(* CODESYS project ccssim.library
   Company: ccsim
   Description: CCS simulator library to support testing tracking devices.
   Version: 0.0.2.0
   Placeholder: ESO CCS PLC Simulator Library
   Author: Mario Kiekebusch
   Title: ESO CCS PLC Simulator Library

Project tree, tasks and I/O mapping:
  libraries: ESO LDC Common Library, * (ESO); ESO LDC Timer Library, * (ESO); Tc2_EtherCAT, * (Beckhoff Automation GmbH); Tc2_IoFunctions, * (Beckhoff Automation GmbH); Tc2_Standard, * (Beckhoff Automation GmbH); Tc2_System, * (Beckhoff Automation GmbH); Tc2_Utilities, * (Beckhoff Automation GmbH); Tc3_Module, * (Beckhoff Automation GmbH); VisuDialogs, * (System); ESO ELT Utility Library, * (ESO)
  DUTs/
    Structures/
      data type T_CCS_CFG
      data type T_CCS_CTRL
      data type T_CCS_GUI
      data type T_CCS_STAT
      data type T_MUDPI_CFG
  GVLs/
    global variables GVL_TrkDefaultEnvironment
    global variables GVL_TrkSiteConstants
  POUs/
    function block FB_CCS_SIM [ST]: FB_init, GetParams, RPC_SetCoordinates, SetParams
    program MAIN [ST]
    program MAIN2 [ST]
  VISUs/
    Templates/
      visualisation GUI_TEMPLATE_CCS_SIM
    visualisation GUI_CCS_SIM
    visualisation GUI_MUDPI_SENDER
    visualisation GUI_TIMER
  text list GlobalTextList
*)

// DUTs/Structures/T_CCS_CFG
TYPE T_CCS_CFG:
STRUCT
	site:     TrkSiteConstants;
	mudpi:    T_MUDPI_CFG;
	ip_address:  Tc2_System.T_IPv4Addr := '192.168.1.2';
END_STRUCT
END_TYPE

// DUTs/Structures/T_CCS_CTRL
TYPE T_CCS_CTRL:
STRUCT
	meanCoordinates: TrkMeanCoordinates;
	environment:     TrkEnvironment;
	motion:          TrkPolarMotion;
	wavelength:      LREAL := 600;
	dut:             LREAL := 0.0;
	equinox:         LREAL := 2000.0;
END_STRUCT
END_TYPE

// DUTs/Structures/T_CCS_GUI
TYPE T_CCS_GUI :
STRUCT
	alt: LREAL;            //[deg]
	az: LREAL;             //[deg]
	pa: LREAL;             //[deg]
	time_tai: STRING;      //[string]
	lst: LREAL;            //[rad]
	ra: LREAL;             //[rad] to be hms in the future
	dec: LREAL;            //[rad] to be dms in the future
	north_angle: LREAL;     //[deg]
	pupil_angle: LREAL;    //[deg]
END_STRUCT
END_TYPE

// DUTs/Structures/T_CCS_STAT
TYPE T_CCS_STAT:
STRUCT
	data       :        PointingKernelPositions;
	// this struct show the same data with different units
	gui_data   :        T_CCS_GUI;
END_STRUCT
END_TYPE

// DUTs/Structures/T_MUDPI_CFG
TYPE T_MUDPI_CFG :
STRUCT
	enabled : BOOL := FALSE; // True if tracking data is sent via MUDPI protocol
	address : UDINT := 0; // Destination IP address for the data as UDINT
	destination_port: UINT := 10000; // Destination port for the data
	source_port: UINT := 8000; // Destination port for the data
	topic_id: UDINT := 500;      // MUDPI Topic identity
	component_id: UINT := 1;  // MUDPI component identity
END_STRUCT
END_TYPE

// GVLs/GVL_TrkDefaultEnvironment
{attribute 'qualified_only'}
VAR_GLOBAL
	C_HUMIDITY:    LREAL := 50.0;
	C_LAPSERATE:   LREAL := 0.0065;
	C_PRESSURE:    LREAL := 760.0;
	C_TEMPERATURE: LREAL := 20;
END_VAR

// GVLs/GVL_TrkSiteConstants
{attribute 'qualified_only'}
VAR_GLOBAL
	C_HEIGHT    : LREAL := 2648;
	C_LONGITUDE : LREAL := 1.228800386;
	C_LATITUDE  : LREAL := -0.429833092;
END_VAR

// POUs/FB_CCS_SIM
FUNCTION_BLOCK FB_CCS_SIM
VAR_INPUT
	refTimeObj  : REFERENCE TO FB_TIME; 
END_VAR
VAR_OUTPUT
END_VAR
VAR
	{attribute 'OPC.UA.DA' := '1'}
	cfg:				T_CCS_CFG;
	{attribute 'OPC.UA.DA' := '1'}
	ctrl:				T_CCS_CTRL;
	{attribute 'OPC.UA.DA' := '1'}
	stat:				T_CCS_STAT;
	
    // Tracking data structure are defined in C++ module
	{attribute 'OPC.UA.DA' := '0'}
	i_trk_data          AT %I*: PointingKernelPositions;
	
	{attribute 'OPC.UA.DA' := '0'}
	q_ccs_data          AT %Q*: CcsData;
	
	{attribute 'OPC.UA.DA' := '0'}
	q_mean_coordinates  AT %Q*: TrkMeanCoordinates;
	
	{attribute 'OPC.UA.DA' := '0'}
	q_mudpi_cfg  AT %Q*: T_MUDPI_CFG;
	
END_VAR


// Get parameters
GetParams();

// Set parameters
SetParams();

METHOD FB_init : BOOL
VAR_INPUT
	bInitRetains : BOOL; // if TRUE, the retain variables are initialized (warm start / cold start)
	bInCopyCode : BOOL;  // if TRUE, the instance afterwards gets moved into the copy code (online change)
END_VAR

cfg.site.height              := GVL_TrkSiteConstants.C_HEIGHT;
cfg.site.latitude            := GVL_TrkSiteConstants.C_LATITUDE;
cfg.site.longitude           := GVL_TrkSiteConstants.C_LONGITUDE;
cfg.mudpi.enabled 			 := FALSE;
cfg.mudpi.destination_port	 := 10000;
cfg.mudpi.source_port		 := 8000;
cfg.mudpi.address			 := 0;
cfg.mudpi.component_id	     := 500;
cfg.mudpi.topic_id			 := 10;
ctrl.environment.humidity    := GVL_TrkDefaultEnvironment.C_HUMIDITY;
ctrl.environment.lapserate   := GVL_TrkDefaultEnvironment.C_LAPSERATE;
ctrl.environment.pressure    := GVL_TrkDefaultEnvironment.C_PRESSURE;
ctrl.environment.temperature := GVL_TrkDefaultEnvironment.C_TEMPERATURE;
ctrl.meanCoordinates.alpha   := 0;
ctrl.meanCoordinates.delta   := -890000.0;
ctrl.meanCoordinates.equinox := 2000.0;
END_METHOD

METHOD GetParams
VAR_INPUT
END_VAR

// Assign output variables according input configuration and control.
memcpy(ADR(q_ccs_data.site), ADR(cfg.site), SIZEOF(q_ccs_data.site));	
memcpy(ADR(q_mudpi_cfg), ADR(cfg.mudpi), SIZEOF(q_mudpi_cfg));	
memcpy(ADR(q_ccs_data.environment), ADR(ctrl.environment), SIZEOF(q_ccs_data.environment));
memcpy(ADR(q_mean_coordinates), ADR(ctrl.meanCoordinates), SIZEOF(q_mean_coordinates));
q_ccs_data.equinox := ctrl.equinox;
q_ccs_data.dut := ctrl.dut;
q_ccs_data.wavelength := ctrl.wavelength;
q_mudpi_cfg.address := F_IpAddress2Integer(IpAddress := cfg.ip_address);
END_METHOD

{attribute 'TcRpcEnable':='1'}
METHOD RPC_SetCoordinates : BOOL
VAR_INPUT
	in_alpha:	 LREAL := 000000.0;
	in_delta:    LREAL := 000000.0;
	in_equinox:  LREAL := 2000.0;
END_VAR

ctrl.meanCoordinates.alpha := in_alpha;
ctrl.meanCoordinates.delta := in_delta;
ctrl.meanCoordinates.equinox := in_equinox;
END_METHOD

METHOD SetParams
VAR_INPUT
END_VAR

//memcpy(ADR(stat.apparent), ADR(i_trk_data.apparent), SIZEOF(stat.apparent));
//memcpy(ADR(stat.observed), ADR(i_trk_data.observed), SIZEOF(stat.observed));
memcpy(ADR(stat.data), ADR(i_trk_data), SIZEOF(stat.data));
stat.gui_data.alt := RAD_TO_DEG(stat.data.target_observed_altaz[0]);
stat.gui_data.az := RAD_TO_DEG(stat.data.target_observed_altaz[1]);
stat.gui_data.pa := RAD_TO_DEG(stat.data.parallactic_angle);
stat.gui_data.ra := F_Rad2Hms(stat.data.radec_at_altaz_at_requested_xy[0]);
stat.gui_data.dec := F_Rad2Dms(stat.data.radec_at_altaz_at_requested_xy[1]);
stat.gui_data.north_angle := RAD_TO_DEG(stat.data.north_angle);
stat.gui_data.pupil_angle := RAD_TO_DEG(stat.data.pupil_angle);
stat.gui_data.time_tai := DCTIME64_TO_STRING(refTimeObj.MudpiTimeToDc(stat.data.time_tai));
END_METHOD

END_FUNCTION_BLOCK

// POUs/MAIN
PROGRAM MAIN
VAR
	ccs_sim:	FB_CCS_SIM;
	fbTimer: FB_TIME;
	diff: LREAL;
END_VAR

fbTimer();
//fbTimer.SetMode(E_TIME_MODE.UTC_NTP);
ccs_sim(refTimeObj := fbTimer);
diff := fbTimer.stat.lrTaiUnixTimeinSecs - ccs_sim.i_trk_data.time_tai;
//ccs_sim.stat.gui_data.time_tai := DCTIME64_TO_STRING(fbTimer.MudpiTimeToDc(ccs_sim.stat.data.time_tai));

END_PROGRAM

// POUs/MAIN2
PROGRAM MAIN2
VAR
	
	fbSender: FB_MUDPI_SENDER;
	
	{attribute 'OPC.UA.DA' := '0'}
	i_trk_data          AT %I*: PointingKernelPositions;
	
END_VAR



fbSender();
fbSender.SetTimestamp(i_trk_data.time_tai);
fbSender.SetMudpiPayload(ADR(i_trk_data), SIZEOF(i_trk_data));
fbSender.SendData();

END_PROGRAM

// VISUs/Templates/GUI_TEMPLATE_CCS_SIM
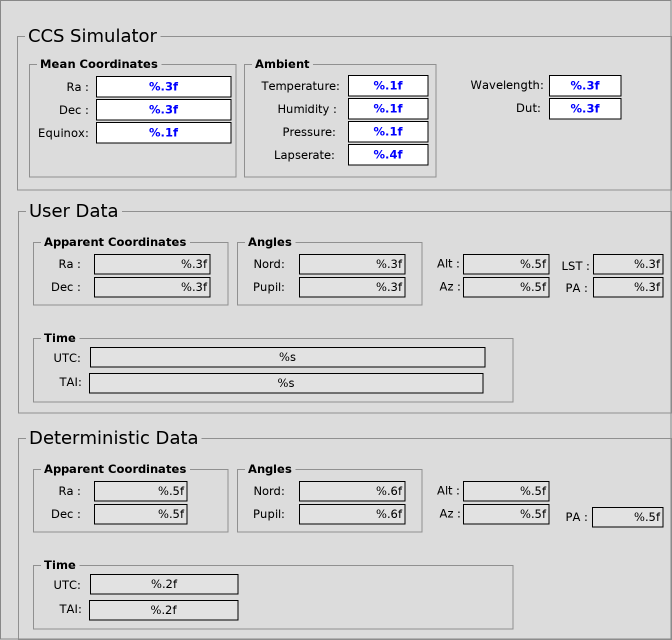
VISUALIZATION GUI_TEMPLATE_CCS_SIM  // 672x640
VAR_INPUT
	m_DeviceName : STRING;
END_VAR
VAR_IN_OUT
	m_Instance : FB_CCS_SIM;
END_VAR
    GroupBox (17,28 655x162), "CCS Simulator"
        GroupBox (12,28 207x121), "Mean Coordinates"
            Label (23,21 40x20), "Ra :"
            Label (23,44 40x20), "Dec :"
            Rectangle (67,20 135x21), "%.3f", tooltip "Mean Right Ascension [hhmmss]", text variable: m_Instance.ctrl.meanCoordinates.alpha
                OnMouseDown: write the text variable via Edit
            Rectangle (67,43 135x21), "%.3f", tooltip "Mean Declination [ddmmss]", text variable: m_Instance.ctrl.meanCoordinates.delta
                OnMouseDown: write the text variable via Edit
            Rectangle (67,66 135x21), "%.1f", tooltip "Equinox", text variable: m_Instance.ctrl.meanCoordinates.equinox
                OnMouseDown: write the text variable via Edit
            Label (3,67 60x20), "Equinox:"
        GroupBox (227,28 192x121), "Ambient"
            Label (7,20 92x20), "Temperature:"
            Label (17,43 79x20), "Humidity :"
            Rectangle (104,19 80x21), "%.1f", tooltip "Temperature [degC]", text variable: m_Instance.ctrl.environment.temperature
                OnMouseDown: write the text variable via Edit
            Rectangle (104,42 80x21), "%.1f", tooltip "Humidity [%]", text variable: m_Instance.ctrl.environment.humidity
                OnMouseDown: write the text variable via Edit
            Rectangle (104,65 80x21), "%.1f", tooltip "Pressure [mbar]", text variable: m_Instance.ctrl.environment.pressure
                OnMouseDown: write the text variable via Edit
            Label (25,66 70x20), "Pressure:"
            Label (24,89 70x20), "Lapserate:"
            Rectangle (104,88 80x21), "%.4f", tooltip "Lapse Rate", text variable: m_Instance.ctrl.environment.lapserate
                OnMouseDown: write the text variable via Edit
        Rectangle (532,47 72x21), "%.3f", text variable: m_Instance.ctrl.wavelength
            OnMouseDown: write the text variable via Edit
        Rectangle (532,70 72x21), "%.3f", text variable: m_Instance.ctrl.dut
            OnMouseDown: write the text variable via Edit
        Label (481,70 46x20), "Dut:"
    GroupBox (18,203 654x210), "User Data"
        GroupBox (15,31 195x71), "Apparent Coordinates"
            Label (11,20 40x20), "Ra :"
            Label (11,43 40x20), "Dec :"
            Label (8,70 60x20)
            Rectangle (61,43 116x20), "%.3f", tooltip "Apparent Declination [ddmmss]", text variable: m_Instance.stat.gui_data.dec
            Rectangle (61,20 116x20), "%.3f", tooltip "Apparent Right Ascension [hhmmss]", text variable: m_Instance.stat.gui_data.ra
        Rectangle (575,74 70x20), "%.3f", tooltip "Parallactic Angle [deg]", text variable: m_Instance.stat.gui_data.pa
        Label (523,75 50x20), "PA :"
        Label (408,51 37x19), "Alt :"
        Label (411,74 35x19), "Az :"
        GroupBox (219,31 185x71), "Angles"
            Label (11,20 40x20), "Nord:"
            Label (11,43 40x20), "Pupil:"
            Label (8,70 60x20)
            Rectangle (62,20 106x20), "%.3f", tooltip "North angle [deg]", text variable: m_Instance.stat.gui_data.north_angle
            Rectangle (62,43 106x20), "%.3f", tooltip "Pupil angle[deg]", text variable: m_Instance.stat.gui_data.pupil_angle
        Rectangle (445,74 86x20), "%.5f", tooltip "TEL Azimuth [deg]", text variable: m_Instance.stat.gui_data.az
        Rectangle (445,51 86x20), "%.5f", tooltip "TEL Altitude [deg]", text variable: m_Instance.stat.gui_data.alt
        GroupBox (15,127 480x72), "Time"
            Label (11,18 40x20), "UTC:"
            Label (6,42 46x20), "TAI:"
            Label (8,70 60x20)
            Rectangle (57,17 395x20), "%s", tooltip "UTC time [sec]", text variable: m_Instance.refTimeObj.stat.sUtcTime
            Rectangle (56,43 394x20), "%s", tooltip "TAI time [sec]", text variable: m_Instance.refTimeObj.stat.sTaiTime
    Label (464,75 83x20), "Wavelength:"
    Label (552,256 41x20), "LST :"
    Rectangle (593,254 70x20), "%.3f", tooltip "Local Sidereal Time [h]", text variable: m_Instance.stat.gui_data.lst
    GroupBox (18,430 654x210), "Deterministic Data"
        GroupBox (15,31 195x71), "Apparent Coordinates"
            Label (11,20 40x20), "Ra :"
            Label (11,43 40x20), "Dec :"
            Label (8,70 60x20)
            Rectangle (61,43 93x20), "%.5f", tooltip "Apparent Declination [rad]", text variable: m_Instance.stat.data.radec_at_altaz_at_requested_xy[1]
            Rectangle (61,20 93x20), "%.5f", tooltip "Apparent Right Ascension [rad]", text variable: m_Instance.stat.data.radec_at_altaz_at_requested_xy[0]
        Rectangle (574,77 71x20), "%.5f", tooltip "Parallactic Angle [rad]", text variable: m_Instance.stat.data.parallactic_angle
        Label (523,77 50x20), "PA :"
        Label (408,51 37x19), "Alt :"
        Label (411,74 35x19), "Az :"
        GroupBox (219,31 185x71), "Angles"
            Label (11,20 40x20), "Nord:"
            Label (11,43 40x20), "Pupil:"
            Label (8,70 60x20)
            Rectangle (62,20 106x20), "%.6f", tooltip "North angle [rad]", text variable: m_Instance.stat.data.north_angle
            Rectangle (62,43 106x20), "%.6f", tooltip "Pupil angle[rad]", text variable: m_Instance.stat.data.pupil_angle
        Rectangle (445,74 86x20), "%.5f", tooltip "TEL Azimuth [rad]", text variable: m_Instance.stat.data.current_observed_altaz[1]
        Rectangle (445,51 86x20), "%.5f", tooltip "TEL Altitude [rad]", text variable: m_Instance.stat.data.current_observed_altaz[0]
        GroupBox (15,127 480x72), "Time"
            Label (11,18 40x20), "UTC:"
            Label (6,42 46x20), "TAI:"
            Label (8,70 60x20)
            Rectangle (57,17 148x20), "%.2f", tooltip "UTC time [sec]", text variable: m_Instance.stat.data.time_utc
            Rectangle (56,43 149x20), "%.2f", tooltip "TAI time [sec]", text variable: m_Instance.stat.data.time_tai
END_VISUALIZATION

// VISUs/GUI_CCS_SIM
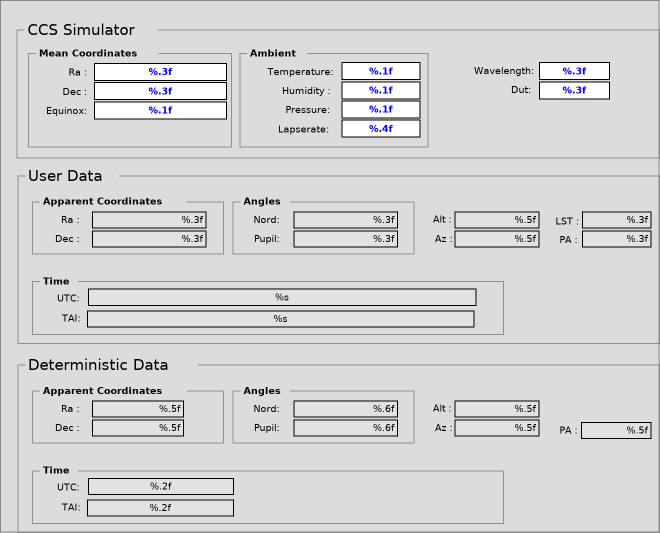
VISUALIZATION GUI_CCS_SIM  // 660x533
    Frame (0,0 660x533)
        shows GUI_TEMPLATE_CCS_SIM(m_DeviceName := ccssim, m_Instance := MAIN.ccs_sim)
END_VISUALIZATION

// VISUs/GUI_MUDPI_SENDER
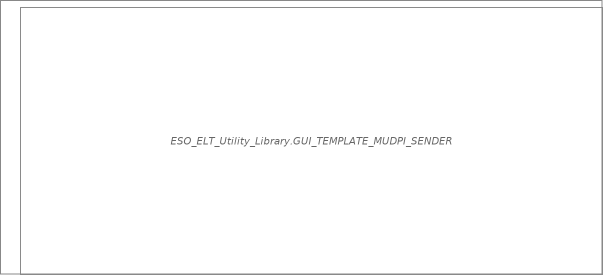
VISUALIZATION GUI_MUDPI_SENDER  // 603x275
    Frame (20,7 583x268)
        shows ESO_ELT_Utility_Library.GUI_TEMPLATE_MUDPI_SENDER(m_Instance := MAIN2.fbSender)
END_VISUALIZATION

// VISUs/GUI_TIMER
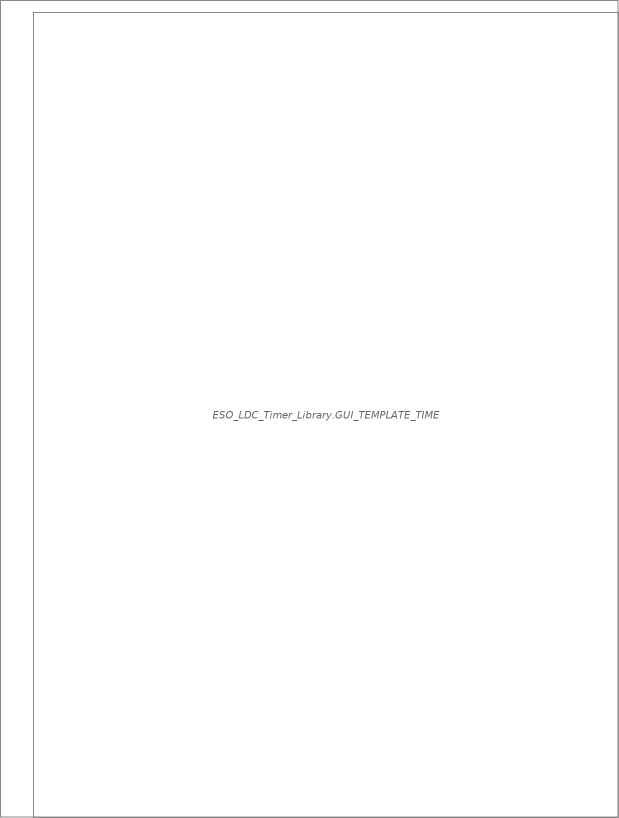
VISUALIZATION GUI_TIMER  // 619x818
    Frame (33,12 586x806)
        shows ESO_LDC_Timer_Library.GUI_TEMPLATE_TIME(m_Instance := MAIN.fbTimer)
END_VISUALIZATION
